Yaskawa INFORM job: JOBDONE.JBI

/JOB
//NAME JOBDONE
//POS
///NPOS 0,0,0,0,0,0
//INST
///DATE 2018/11/28 11:02
///ATTR SC,RW,MC
NOP
DOUT OT#(594) OFF
TIMER T=0.50
WAIT IG#(78)=0
WAIT IG#(77)=0
DOUT OT#(595) ON
WAIT IN#(595)=ON
DOUT OT#(595) OFF
END
